// TIA Portal project "Modbus" (V15.1)

(* hardware
DEVICE "S71500/ET200MP station_1"  S7-1500 station
   slot 0: "Rail_0"  Rack  6ES7 590-1***0-0AA0
   slot 1: "PLC_1"  CPU 1511C-1 PN  6ES7 511-1CK01-0AB0  V2.6
      slot 3: "CPU display_1"  6ES7591-1AA00-0AA0
   slot 2: "CM PtP RS422/485 BA_1"  CM PtP RS422/485 BA  6ES7 540-1AB00-0AA0  V1.0
*)

// ===== PLC "PLC_1"  CPU 1511C-1 PN =====

TYPE "modbusCommLoad"
   STRUCT
      Done : Bool;
      Error : Bool;
      Status : Word;
      ErrorStatus : Word;
      DoneStored : Bool;
   END_STRUCT;
END_TYPE

TYPE "modbusMasterCmd"
   STRUCT
      req : Bool;
      MbAddr : UInt;
      Mode : USInt;
      DataAddr : UDInt;
      DataLen : UInt;
      Done : Bool;
      Busy : Bool;
      Error : Bool;
      Status : Word;
      ErrorStatus : Word;
   END_STRUCT;
END_TYPE

TYPE "modbusSlaveCmd"
   STRUCT
      MbAddr : UInt;
      MbHoldReg : Word;
      Ndr : Bool;
      Dr : Bool;
      Error : Bool;
      Status : Word;
   END_STRUCT;
END_TYPE

DATA_BLOCK "Output_Data"   // DB3
{ S7_Optimized_Access := 'TRUE' }
VERSION : 0.1
BEGIN
END_DATA_BLOCK

DATA_BLOCK "Comm_Data"   // DB4
{ S7_Optimized_Access := 'TRUE' }
VERSION : 0.1
BEGIN
END_DATA_BLOCK

DATA_BLOCK "Process"   // DB6
{ S7_Optimized_Access := 'TRUE' }
VERSION : 0.1
   VAR
      "step" : USInt;
      modbusCommLoad : "modbusCommLoad";
      modbusMasterCmd : "modbusMasterCmd";
      modbusSlaveCmd : "modbusSlaveCmd";
   END_VAR
BEGIN
END_DATA_BLOCK

DATA_BLOCK "MasterData"   // DB7
{ S7_Optimized_Access := 'TRUE' }
VERSION : 0.1
   VAR
      DataPtr : Word;
   END_VAR
BEGIN
END_DATA_BLOCK

ORGANIZATION_BLOCK "Main"   // OB1, LAD, ProgramCycle
TITLE = "Main Program Sweep (Cycle)"
{ S7_Optimized_Access := 'TRUE' }
VERSION : 0.1
   VAR_INPUT
      Initial_Call : Bool;   // Initial call of this OB
      Remanence : Bool;   // =True, if remanent data are available
   END_VAR
BEGIN

REGION Network 1: Configuración para establecer comunicación
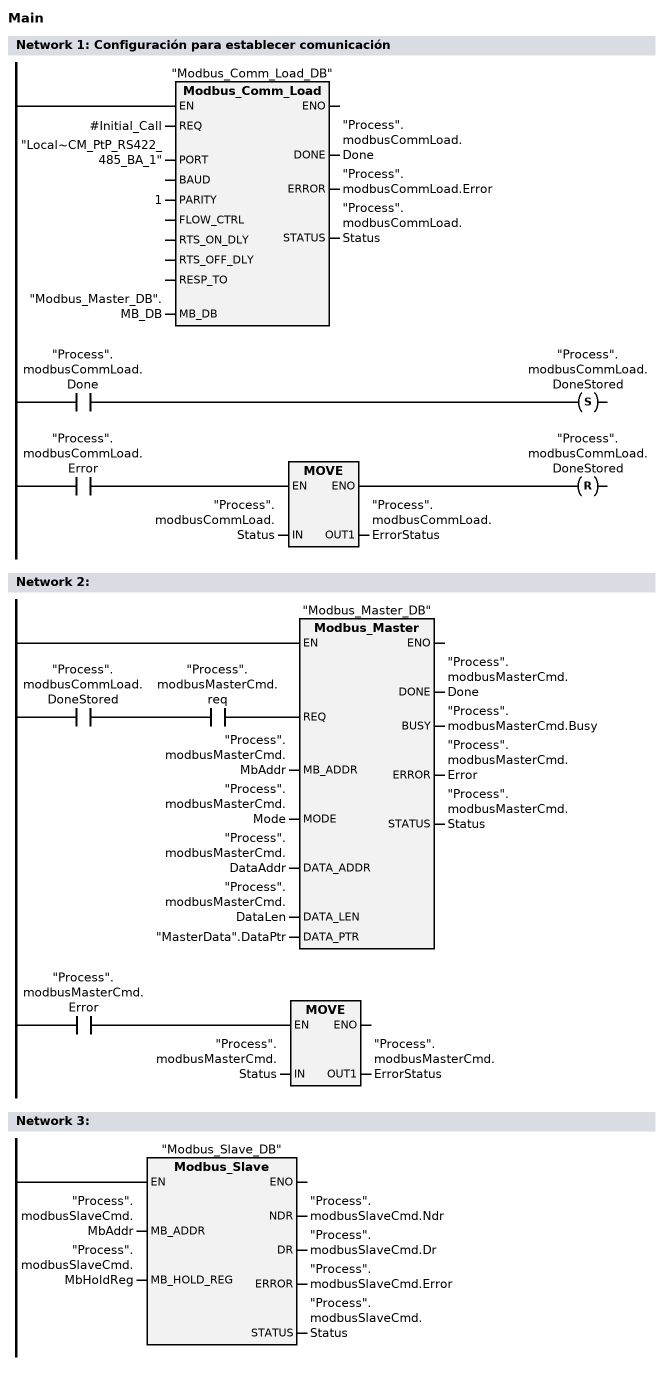
   "Modbus_Comm_Load_DB"(REQ := #Initial_Call,   // Modbus_Comm_Load
                         PORT := "Local~CM_PtP_RS422_485_BA_1",
                         PARITY := 1,
                         MB_DB := "Modbus_Master_DB".MB_DB,
                         DONE => "Process".modbusCommLoad.Done,
                         ERROR => "Process".modbusCommLoad.Error,
                         STATUS => "Process".modbusCommLoad.Status);
   IF "Process".modbusCommLoad.Done THEN "Process".modbusCommLoad.DoneStored := TRUE; END_IF;
   IF "Process".modbusCommLoad.Error THEN
       "Process".modbusCommLoad.ErrorStatus := "Process".modbusCommLoad.Status;
       "Process".modbusCommLoad.DoneStored := FALSE;
   END_IF;
END_REGION

REGION Network 2
   "Modbus_Master_DB"(REQ := "Process".modbusCommLoad.DoneStored AND "Process".modbusMasterCmd.req,   // Modbus_Master
                      MB_ADDR := "Process".modbusMasterCmd.MbAddr,
                      MODE := "Process".modbusMasterCmd.Mode,
                      DATA_ADDR := "Process".modbusMasterCmd.DataAddr,
                      DATA_LEN := "Process".modbusMasterCmd.DataLen,
                      DATA_PTR := "MasterData".DataPtr,
                      DONE => "Process".modbusMasterCmd.Done,
                      BUSY => "Process".modbusMasterCmd.Busy,
                      ERROR => "Process".modbusMasterCmd.Error,
                      STATUS => "Process".modbusMasterCmd.Status);
   IF "Process".modbusMasterCmd.Error THEN
       "Process".modbusMasterCmd.ErrorStatus := "Process".modbusMasterCmd.Status;
   END_IF;
END_REGION

REGION Network 3
   "Modbus_Slave_DB"(MB_ADDR := "Process".modbusSlaveCmd.MbAddr,   // Modbus_Slave
                     MB_HOLD_REG := "Process".modbusSlaveCmd.MbHoldReg,
                     NDR => "Process".modbusSlaveCmd.Ndr,
                     DR => "Process".modbusSlaveCmd.Dr,
                     ERROR => "Process".modbusSlaveCmd.Error,
                     STATUS => "Process".modbusSlaveCmd.Status);
END_REGION
END_ORGANIZATION_BLOCK